{attribute 'linkalways'} 
{attribute 'no_explicit_call' := 'This FB is a CLASS and must be accessed using methods or properties'}
{attribute 'enable_dynamic_creation'}
FUNCTION_BLOCK _LINT EXTENDS NumericDatatypeBase
VAR
	localData : LINT;
	activeData : REFERENCE TO LINT REF= localData;
END_VAR

PROPERTY PUBLIC Address : PVOID
GET
Address := ADR(activeData);
END_GET
END_PROPERTY

METHOD PUBLIC ClearReference
VAR_INPUT
END_VAR
activeData REF= localData;
END_METHOD

METHOD PUBLIC Clone : I_Datatype
VAR
    pClone : POINTER TO _LINT;
END_VAR
pClone := __NEW(_LINT(InitialValue := Value));
Clone := pClone^;
END_METHOD

METHOD FB_init : BOOL
VAR_INPUT
	bInitRetains : BOOL; // if TRUE, the retain variables are initialized (warm start / cold start)
	bInCopyCode : BOOL;  // if TRUE, the instance afterwards gets moved into the copy code (online change)
	InitialValue : LINT;
END_VAR
localData := InitialValue;
END_METHOD

PROPERTY PUBLIC IsFloat : BOOL
GET
IsFloat := FALSE;
END_GET
END_PROPERTY

PROPERTY PUBLIC IsSigned : BOOL
GET
IsSigned := TRUE;
END_GET
END_PROPERTY

METHOD PUBLIC MakeReferenceTo
VAR_INPUT
	ReferenceTarget : REFERENCE TO LINT;
END_VAR
activeData REF= ReferenceTarget;
END_METHOD

PROPERTY PUBLIC MaxValue : LINT
GET
MaxValue :=  DatatypeLimits.LINT_MAX_VALUE;
END_GET
END_PROPERTY

PROPERTY PUBLIC MinValue : LINT
GET
MinValue := DatatypeLimits.LINT_MIN_VALUE;
END_GET
END_PROPERTY

METHOD PROTECTED SerializeMaxValue
VAR_INPUT
	Serializer : I_Serializer;
END_VAR
Serializer.AddLint(MaxValue);
END_METHOD

METHOD PROTECTED SerializeMinValue
VAR_INPUT
	Serializer : I_Serializer;
END_VAR
Serializer.AddLint(MinValue);
END_METHOD

METHOD PUBLIC SerializeWith
VAR_INPUT
	Serializer : I_Serializer;
END_VAR
Serializer.AddLint(activeData);
END_METHOD

PROPERTY PUBLIC Size : UDINT
GET
Size := SIZEOF(activeData);
END_GET
END_PROPERTY

METHOD TryDeserializeFrom : BOOL
VAR_INPUT
	Deserializer : I_Deserializer;
	Feedback : I_DeserializerFeedback;
END_VAR
TryDeserializeFrom := Deserializer.TryGetLint(activeData, Feedback);
END_METHOD

METHOD TryMakeReferenceTo : BOOL
VAR_INPUT
	Target : I_Datatype;
END_VAR
VAR
	pTargetData : POINTER TO LINT;
END_VAR
IF NOT (Target.TypeName = TypeName) THEN
	RETURN;
END_IF

pTargetData := Target.Address;
activeData REF= pTargetData^;
TryMakeReferenceTo := TRUE;
END_METHOD

PROPERTY PUBLIC TypeName : T_MAXSTRING
GET
TypeName := 'LINT';
END_GET
END_PROPERTY

PROPERTY PUBLIC Value : LINT
GET
Value := activeData;
END_GET
SET
activeData := Value;
END_SET
END_PROPERTY

END_FUNCTION_BLOCK

(* stored: Version 1.1.0.1, ProductVersion 3.1.4024.12
   POU _LINT: Id {fd3f17c8-3c55-4be4-967b-a6f1ccfb45aa}, SpecialFunc None
   Folder Constructor: Id {0ddbc8d5-6d77-43d8-92d9-2582a83fd528}
   Folder Protected: Id {d1baa519-0fa5-4cd8-b580-4a510dd0a033}
   Property Address: Id {a607453a-554d-4afe-ac58-c98463e0175b}
   Get Get: Id {95726774-34a6-43c5-8b30-914840367b36}
   Method ClearReference: Id {ad44e6b3-8387-426c-9fb1-f2c663dd3e48}
   Method Clone: Id {06190932-46b7-49e9-98a7-70afb27671e2}
   Method FB_init: Id {85dc6098-a22e-4705-be6f-117581307a4f}
   Property IsFloat: Id {47ce383c-e837-48d8-b3b1-b3b909b78fd8}
   Get Get: Id {4f3d39f6-3bb4-4f8b-9378-e1275cdf8182}
   Property IsSigned: Id {43b63b9c-b5cb-4a92-aca8-66dc4360c4fd}
   Get Get: Id {ac616a1c-8c86-4d91-9a24-4fb376455693}
   Method MakeReferenceTo: Id {c6a71264-fdb3-4123-a49a-cb0bdaf8ed54}
   Property MaxValue: Id {ee0def83-f845-42f1-a62a-f986140db531}
   Get Get: Id {1f9bb036-3d9d-47db-82da-c784d606bfb1}
   Property MinValue: Id {f2c801ca-6638-464e-af23-9c38c9113da5}
   Get Get: Id {071725b4-c7a9-4395-bab6-cb3ad1ad7b98}
   Method SerializeMaxValue: Id {52ef821e-85d9-4b57-8bf9-9f375369e237}
   Method SerializeMinValue: Id {da6b2ed7-3d40-44b8-81ae-8e8f2849ed00}
   Method SerializeWith: Id {a6733c32-0062-451f-9c88-973fcef906ad}
   Property Size: Id {9307ec41-474e-436e-a746-a0f4078f6cd0}
   Get Get: Id {24ba2fec-737b-4135-a8da-d3d0d550493b}
   Method TryDeserializeFrom: Id {40bde53e-6ce9-4722-b5d0-6d3585ca1778}
   Method TryMakeReferenceTo: Id {a8627b2b-02e0-454b-b63a-51bf85a468aa}
   Property TypeName: Id {477dbe68-2638-4e48-abcf-399e45441b9a}
   Get Get: Id {9316f4af-61df-4dcf-b14d-667d55e0052a}
   Property Value: Id {2f76c94a-9b8d-48e1-a4a9-25a018e053aa}
   Get Get: Id {981252d6-ddcd-4477-9b18-ac4de4223bf3}
   Set Set: Id {60c66633-bad6-42ed-9053-2cbb5864b9ee} *)
